Yaskawa INFORM job: WELDING-CMF100-ST1-FRONT.JBI

/JOB
//NAME WELDING-CMF100-ST1-FRONT
//POS
///NPOS 16,16,16,1,0,0
///TOOL 0
///POSTYPE PULSE
///PULSE
C00000=-135635,-48720,-26872,-24315,58563,60510
C00001=-164109,-31285,-43199,-96851,54836,104336
C00002=-156495,-6630,-44443,-130972,44695,123587
C00003=-157047,10945,-56859,-142614,18847,130779
C00004=-157047,10640,-56731,-142578,19068,130721
C00005=-156844,10346,-56984,-142715,19089,130779
C00006=-155545,-5827,-29336,-112145,57583,112738
C00007=-155505,-5835,-29287,-112123,57624,112718
C00008=-155515,-5815,-29329,-112176,57599,112754
C00009=-155514,-5834,-29248,-112072,57633,112686
C00010=-151780,5203,886,-48753,60896,77150
C00011=-147433,45315,64682,-14232,30892,56744
C00012=-134548,56882,84835,-4380,21141,50689
C00013=-148229,-2526,1565,-46439,64385,76694
C00014=-127230,-32198,-22151,-29001,72518,65896
C00015=-125474,-40572,-24853,-5768,46716,52915
BC00000=246221
BC00001=276929
BC00002=276929
BC00003=276929
BC00004=276929
BC00005=276929
BC00006=276929
BC00007=276929
BC00008=276929
BC00009=276929
BC00010=276929
BC00011=276929
BC00012=247202
BC00013=276929
BC00014=276929
BC00015=272147
EC00000=2040560
EC00001=2040560
EC00002=2040560
EC00003=2302582
EC00004=2302582
EC00005=2302582
EC00006=2016830
EC00007=1029563
EC00008=-3664
EC00009=-1005635
EC00010=-1331629
EC00011=-1504884
EC00012=-1546557
EC00013=-1471191
EC00014=-1051894
EC00015=-573101
///USER 10
///POSTYPE USER
///RECTAN
///RCONF 0,0,0,0,0,0,0,0,0,0,0,0,0,0,0,0,0,0,0,0,0,0,0,0
P00049=2.600,0.000,0.000,0.0000,0.0000,0.0000
//INST
///DATE 2018/10/04 11:52
///ATTR SC,RW
///GROUP1 RB1,BS1
///GROUP2 ST1
NOP
'***** welding station 1 front
MOVJ C00000 BC00000 VJ=25.00  +MOVJ EC00000 VJ=100.00
'***** go to start pos
SMOVL C00001 BC00001 V=166.7 PL=0  +MOVJ EC00001
SFTON P049 UF#(10)
SMOVL C00002 BC00002 V=83.3  +MOVJ EC00002
SMOVC C00003 BC00003 V=83.3 PL=0  +MOVJ EC00003  //start welding
DOUT OT#(656) OFF
TIMER T=0.50
DOUT OT#(656) ON
DOUT OT#(46) ON
DOUT OT#(45) ON
DOUT OT#(46) ON
MACRO1 MJ#(5) ARGF3
SREFP 1 C00004 BC00004  +REFP EC00004
SREFP 2 C00005 BC00005  +REFP EC00005
ARCON ASF#(1)
SWVON WEV#(1)
SMOVC C00006 BC00006 V=I000  +MOVJ EC00006
SMOVC C00007 BC00007 V=I000  +MOVJ EC00007
SMOVC C00008 BC00008 V=I000  +MOVJ EC00008
SMOVC C00009 BC00009 V=I000  +MOVJ EC00009
SMOVC C00010 BC00010 V=I000  +MOVJ EC00010
SMOVC C00011 BC00011 V=I000  +MOVJ EC00011
ARCOF
SMOVL C00012 BC00012 V=I000  +MOVJ EC00012
MACRO1 MJ#(5) ARGF5
DOUT OT#(656) OFF
SWVOF
TIMER T=5.00
'***** go to end position
SMOVL C00013 BC00013 V=83.3 PL=0  +MOVJ EC00013
SMOVL C00014 BC00014 V=83.3  +MOVJ EC00014
MOVL C00015 BC00015 V=166.7  +MOVJ EC00015 VJ=100.00
END
